{attribute addProperty BoxType "EL6002-0000-0017"}
{attribute addProperty Id "StatusAT %I*Status_0CBEDEF81621Data_InAT %I*ARRAY[0 ..21] OF USINT176220"}
{attribute addProperty CRC "3699519399"}
{attribute addProperty SizeInBites "192"}
{attribute addProperty SizeInBytes "24"}
TYPE COM_TxPDO_Map_Inputs_Channel_85D1D733 :
STRUCT
	{attribute addProperty Name "Status"}
	Status AT %I* : Status_0CBEDEF8;
	{attribute addProperty Name "Data_In"}
	Data_In AT %I* : ARRAY[0 ..21] OF USINT;
END_STRUCT
END_TYPE

(* stored: Version 1.2.0.0, ProductVersion 3.1.4024.9
   DUT COM_TxPDO_Map_Inputs_Channel_85D1D733: Id {d6001dc2-4c50-4e68-b1cd-ba85a816a181} *)
